TYPE SAFETY_OUT :
STRUCT

	DOORS_RUN:BOOL;
	DOORS_ErrAck:BOOL;

	NOT_AUS_RUN:BOOL;
	NOT_AUS_ErrAck:BOOL;

	NOT_AUS_RESET:BOOL;

END_STRUCT
END_TYPE

(* stored: Version 1.1.0.1, ProductVersion 3.1.0.26
   DUT SAFETY_OUT: Id {f20ccb0f-d85a-4d62-a80f-23bfc90c5ddc} *)
